PROGRAM prgGrid
VAR
	lrPowerGridkW		: LREAL;	//{#lynus.ag#()}
END_VAR

lrPowerGridkW := prgPV.lrPowerHouse - prgPV.lrPowerPV;

END_PROGRAM

(* stored: Version 1.1.0.1, ProductVersion 3.1.4024.9
   POU prgGrid: Id {1288d895-13e1-4c5e-ac38-ff2df2ce2ff9}, SpecialFunc None *)
